TYPE TPhaseHeating :
STRUCT
	Cmd : TPhaseCmd;
	State : TPhaseState;
	
	ParamReqTemp : REAL;
	
	WaterTemp : REAL;
	
	fTime : INT;
END_STRUCT
END_TYPE

(* stored: Version 1.1.0.1, ProductVersion 3.1.4024.13
   DUT TPhaseHeating: Id {25440770-ac65-42dd-8945-2dbb24707357} *)
